{attribute 'linkalways'} 
{attribute 'no_explicit_call' := 'This FB is a CLASS and must be accessed using methods or properties'}
{attribute 'enable_dynamic_creation'}
FUNCTION_BLOCK OrderedDictionary EXTENDS Disposable IMPLEMENTS I_Dictionary
VAR
	eventEmitter : EventEmitter;
	rootNode : I_OrderedDictionaryTreeNode;
	head : I_OrderedDictionaryTreeNode;
	tail : I_OrderedDictionaryTreeNode;
END_VAR

METHOD PRIVATE AddKeysInOrderToCollection
VAR_INPUT
	Collection : I_Collection;
END_VAR
VAR
	currentNode : I_OrderedDictionaryTreeNode;
	key : T_MAXSTRING;
END_VAR
IF head = 0 THEN
	RETURN;
END_IF

currentNode := head;

REPEAT
    key := currentNode.Key;
	Collection.AddItem(key);
	currentNode := currentNode.Next;
UNTIL
    currentNode = 0
END_REPEAT;
END_METHOD

METHOD PRIVATE AddNodesInOrderToCollection
VAR_INPUT
	Collection : I_Collection;
END_VAR
VAR
	currentNode : I_OrderedDictionaryTreeNode;
	key : T_MAXSTRING;
END_VAR
IF head = 0 THEN
	RETURN;
END_IF

currentNode := head;

REPEAT
	Collection.AddItem(currentNode);
	currentNode := currentNode.Next;
UNTIL
    currentNode = 0
END_REPEAT;
END_METHOD

METHOD PRIVATE AddNodeToEnd
VAR_INPUT
	Node : I_OrderedDictionaryTreeNode;
END_VAR
VAR
	originalTailNode : I_OrderedDictionaryTreeNode;
END_VAR
//LogMsg_I_OrderedDictionaryTreeNode('OrderedDictionary', 'AddNodeToEnd: Called with', Node);

IF head = 0 THEN
	head := Node;
	tail := Node;
	Node.Previous := 0;
	Node.Next := 0;
//	LogMsg('OrderedDictionary', 'AddNodeToEnd: Return, head = 0');
//	LogMsg_I_OrderedDictionaryTreeNode('OrderedDictionary', 'AddNodeToEnd: Head is', head);
//	LogMsg_I_OrderedDictionaryTreeNode('OrderedDictionary', 'AddNodeToEnd: Tail is', tail);
	RETURN;
END_IF

//LogMsg_I_OrderedDictionaryTreeNode('OrderedDictionary', 'AddNodeToEnd: Original Tail was', tail);
originalTailNode := tail;
tail := Node;
//LogMsg_I_OrderedDictionaryTreeNode('OrderedDictionary', 'AddNodeToEnd: Tail is now', tail);

originalTailNode.Next := node;
//LogMsg_I_OrderedDictionaryTreeNode('OrderedDictionary', 'AddNodeToEnd: Original Tail next is', originalTailNode.Next);
tail.Previous := originalTailNode;
tail.Next := 0;
//LogMsg_I_OrderedDictionaryTreeNode('OrderedDictionary', 'AddNodeToEnd: Tail previous is now', tail.Previous);

//LogMsg('OrderedDictionary', 'AddNodeToEnd: Return');
END_METHOD

METHOD PUBLIC AddOrUpdate
VAR_INPUT
	Key : T_MAXSTRING;
	Value : ANY;
END_VAR
rootNode := THIS^.RecursiveInsert(Key, Value, rootNode);
EmitChangedEvent();
END_METHOD

METHOD PRIVATE Balance : I_OrderedDictionaryTreeNode
VAR_INPUT
	Node : I_OrderedDictionaryTreeNode;
END_VAR
VAR
	balanceFactor : DINT;
END_VAR
balanceFactor := THIS^.GetBalanceFactor(Node);

IF (balanceFactor > 1) THEN
	IF THIS^.GetBalanceFactor(Node.Left) < 0 THEN
		Node.Left := THIS^.LeftRotate(Node.Left);
	END_IF
	Node := RightRotate(Node);
ELSIF (balanceFactor < -1) THEN
	IF THIS^.GetBalanceFactor(Node.Right) > 0 THEN
		Node.Right := RightRotate(Node.Right);
	END_IF
	Node := LeftRotate(Node);
END_IF

Balance := Node;

//LogMsg('OrderedDictionary', ': Called');
//LogMsg_I_OrderedDictionaryTreeNode('OrderedDictionary', ': RootNode is now', rootNode);
//LogMsg('OrderedDictionary', ': Return');
END_METHOD

METHOD PUBLIC Clear
VAR_INPUT
END_VAR
VAR
	currentNode : I_OrderedDictionaryTreeNode;
	nextNode : I_OrderedDictionaryTreeNode;
END_VAR
IF head = 0 THEN
	RETURN;
END_IF

currentNode := head;

WHILE currentNode <> 0 DO
	nextNode := currentNode.Next;
	currentNode.Dispose();
	currentNode := nextNode;
END_WHILE

head := 0;
tail := 0;
rootNode := 0;
EmitChangedEvent();
END_METHOD

METHOD PUBLIC ContainsKey : BOOL
VAR_INPUT
	Key : T_MAXSTRING;
END_VAR
VAR
	foundNode : I_OrderedDictionaryTreeNode;
END_VAR
foundNode := THIS^.RecursiveFind(Key, rootNode);

IF foundNode = 0 THEN
	RETURN;
END_IF

ContainsKey := TRUE;
END_METHOD

PROPERTY PUBLIC Count : DINT
GET
VAR
	NodeCount : DINT;
END_VAR
RecursiveCountNodes(rootNode, NodeCount);
Count := NodeCount;
END_GET
END_PROPERTY

METHOD PRIVATE EmitChangedEvent
VAR
	dictionaryChangedEvent : KeyValueCollectionChangedEvent(Target := THIS^);
END_VAR
eventEmitter.Emit('OnChanged', dictionaryChangedEvent);
END_METHOD

METHOD PRIVATE EmitDisposedEvent
VAR
	dictionaryDisposedEvent : KeyValueCollectionDisposedEvent(Target := THIS^);
END_VAR
eventEmitter.Emit('OnDisposed', dictionaryDisposedEvent);
END_METHOD

METHOD FB_exit : BOOL
VAR_INPUT
	bInCopyCode : BOOL; // if TRUE, the exit method is called for exiting an instance that is copied afterwards (online change).
END_VAR
VAR
END_VAR
IF bInCopyCode THEN
    RETURN;
END_IF

Clear();
EmitDisposedEvent();
END_METHOD

METHOD PRIVATE FindMinimum : I_OrderedDictionaryTreeNode
VAR_INPUT
	Node : I_OrderedDictionaryTreeNode;
END_VAR
VAR
	nextNode : I_OrderedDictionaryTreeNode;
END_VAR
nextNode := Node;

WHILE (nextNode.left <> 0) DO
      nextNode := nextNode.left;
END_WHILE;

FindMinimum := nextNode;
END_METHOD

METHOD PRIVATE GetBalanceFactor : DINT
VAR_INPUT
	Node : I_OrderedDictionaryTreeNode;
END_VAR
IF (Node = 0) THEN
	GetBalanceFactor := 0;
	RETURN;
END_IF

GetBalanceFactor := THIS^.GetHeight(node.left) - THIS^.GetHeight(node.right);
END_METHOD

METHOD GetEnumerator : I_ForwardEnumerator
VAR
	pNodeCollection : POINTER TO LinkedList;
	pEnumerator : POINTER TO OrderedDictionaryForwardEnumerator;
END_VAR
pNodeCollection := __NEW(LinkedList);
THIS^.AddNodesInOrderToCollection(pNodeCollection^);

pEnumerator := __NEW(OrderedDictionaryForwardEnumerator(Parent := THIS^, Nodes := pNodeCollection^));
GetEnumerator := pEnumerator^;
END_METHOD

METHOD PRIVATE GetHeight : DINT
VAR_INPUT
	Node : I_OrderedDictionaryTreeNode;
END_VAR
IF Node = 0 THEN
	GetHeight := -1;
	RETURN;
END_IF

GetHeight := Node.Height;
END_METHOD

METHOD PUBLIC GetKeys : I_Collection
VAR
	pLinkedList : POINTER TO LinkedList;
END_VAR
pLinkedList := __NEW(LinkedList);
THIS^.AddKeysInOrderToCollection(pLinkedList^);
GetKeys := pLinkedList^;
END_METHOD

METHOD GetKeyValueEnumerator : I_KeyValueForwardEnumerator
VAR
	pNodeCollection : POINTER TO LinkedList;
	pEnumerator : POINTER TO OrderedDictionaryForwardEnumerator;
END_VAR
pNodeCollection := __NEW(LinkedList);
THIS^.AddNodesInOrderToCollection(pNodeCollection^);

pEnumerator := __NEW(OrderedDictionaryForwardEnumerator(Parent := THIS^, Nodes := pNodeCollection^));
GetKeyValueEnumerator := pEnumerator^;
END_METHOD

PROPERTY IsEmpty : BOOL
GET
IsEmpty := rootNode = 0;
END_GET
END_PROPERTY

METHOD PRIVATE LeftRotate : I_OrderedDictionaryTreeNode
VAR_INPUT
	X : I_OrderedDictionaryTreeNode;
END_VAR
VAR
	y : I_OrderedDictionaryTreeNode;
	t2 : I_OrderedDictionaryTreeNode;
END_VAR
y := X.right;
t2 := y.left;
y.left := X;
X.right := t2;
THIS^.UpdateHeight(X);
THIS^.UpdateHeight(y);
LeftRotate := y;
END_METHOD

METHOD PUBLIC OffEvent
VAR_INPUT
	EventName : T_MaxString;
	EventHandler : I_EventHandler;
END_VAR
eventEmitter.OffEvent(EventName, EventHandler);
END_METHOD

METHOD PUBLIC OnceEvent
VAR_INPUT
	EventName : T_MaxString;
	EventHandler : I_EventHandler;
END_VAR
eventEmitter.OnceEvent(EventName, EventHandler);
END_METHOD

METHOD PUBLIC OnEvent
VAR_INPUT
	EventName : T_MaxString;
	EventHandler : I_EventHandler;
END_VAR
eventEmitter.OnEvent(EventName, EventHandler);
END_METHOD

METHOD PRIVATE RecursiveCountNodes
VAR_INPUT
	Node : I_OrderedDictionaryTreeNode;
	Count : REFERENCE TO DINT;
END_VAR
IF Node = 0 THEN
	RETURN;
END_IF

Count := Count + 1;

THIS^.RecursiveCountNodes(Node.Left,Count);
THIS^.RecursiveCountNodes(Node.Right,Count);
END_METHOD

METHOD PRIVATE RecursiveDelete : I_OrderedDictionaryTreeNode
VAR_INPUT
	Key : T_MAXSTRING;
	Node : I_OrderedDictionaryTreeNode;
END_VAR
VAR
	newNode : I_OrderedDictionaryTreeNode; 
	minValueNode : I_OrderedDictionaryTreeNode;
	minValueNodeParent : I_OrderedDictionaryTreeNode;
	balanceFactor : DINT;
END_VAR
IF (Node = 0) THEN
    RETURN;
END_IF

IF (Key < Node.Key) THEN
    Node.left := THIS^.RecursiveDelete(Key, Node.left);
ELSIF (Key > Node.Key) THEN
    Node.right := THIS^.RecursiveDelete(Key, Node.right);
ELSE
    IF (Node.Left = 0) OR (Node.Right = 0) THEN
        IF (Node.Left = 0) THEN
            newNode := Node.Right;
        ELSE
            newNode := Node.Left;
        END_IF
		RemoveNodeFromLinkedList(Node);
        Node.Dispose();
        THIS^.updateHeight(newNode);
        RecursiveDelete := THIS^.Balance(newNode);
        RETURN;
    ELSE
		RemoveNodeFromLinkedList(Node);
		minValueNode := FindMinimum(Node.Right);
		ReplaceNodeInLinkedList(minValueNode, Node);
        Node.Right := THIS^.RecursiveDelete(minValueNode.Key, Node.Right);	
    END_IF
END_IF

THIS^.updateHeight(Node);
RecursiveDelete := THIS^.Balance(Node);
END_METHOD

METHOD PRIVATE RecursiveFind : I_OrderedDictionaryTreeNode
VAR_INPUT
	Key : T_MAXSTRING;
	Node : I_OrderedDictionaryTreeNode;
END_VAR
IF (Node = 0) THEN
	RETURN;
END_IF

IF (Key < Node.key) THEN
  RecursiveFind := THIS^.RecursiveFind(key, Node.left);
  RETURN;
ELSIF (key > Node.key) THEN
  RecursiveFind := THIS^.RecursiveFind(key, Node.right);
  RETURN;
ELSE 
  RecursiveFind := Node;
  RETURN;
END_IF
END_METHOD

METHOD PRIVATE RecursiveInsert : I_OrderedDictionaryTreeNode
VAR_INPUT
	Key : T_MAXSTRING;
	Value : ANY;
	Node : I_OrderedDictionaryTreeNode;
END_VAR
VAR
	pAVLTreeNode : POINTER TO OrderedDictionaryTreeNode;
	balanceFactor : DINT;
END_VAR
IF (Node = 0) THEN
	pAVLTreeNode := __NEW(OrderedDictionaryTreeNode(NodeKey := Key, NodeSource := Value));
	AddNodeToEnd(pAVLTreeNode^);
	RecursiveInsert := pAVLTreeNode^;
	RETURN;
END_IF

IF (Key < Node.Key) THEN
	Node.left := THIS^.RecursiveInsert(Key, Value, Node.left);
ELSIF (Key > Node.Key) THEN
	Node.right := THIS^.RecursiveInsert(Key, Value, Node.right);
ELSE
	Node.Reinitialize(Key,Value);
	RecursiveInsert := Node;
END_IF

THIS^.updateHeight(node);

balanceFactor := THIS^.GetBalanceFactor(Node);
Node := balance(Node);
RecursiveInsert := Node;
END_METHOD

METHOD PUBLIC Remove
VAR_INPUT
	Key : T_MAXSTRING;
END_VAR
rootNode := THIS^.RecursiveDelete(Key, rootNode);
EmitChangedEvent();
END_METHOD

METHOD PRIVATE RemoveNodeFromLinkedList
VAR_INPUT
	Node : I_OrderedDictionaryTreeNode;
END_VAR
VAR
	nodeBefore : I_OrderedDictionaryTreeNode; 
	nodeAfter : I_OrderedDictionaryTreeNode;
END_VAR
// if the node is the head and has no further nodes following it, then it must
// be the only node in the collection.  As such, set head, tail as 0.
IF Node = head AND Node = tail THEN
	head := 0;
	tail := 0;
	Node.Previous := 0;
	Node.Next := 0;
	RETURN;
END_IF

// if the node is at the start of more than one node, then
// make the next in line the head, and remove it's knowlege of
// the node being removed.
IF Node = head THEN
	Node.Next.Previous := 0;
	head := Node.Next;
	Node.Previous := 0;
	Node.Next := 0;
	RETURN;
END_IF

// if the node is at the end of more than one node, then
// make the previous in line the tail, and remove it's knowlege of
// the node being removed.
IF Node = tail THEN
	Node.Previous.Next := 0;
	tail := Node.Previous;
	Node.Previous := 0;
	Node.Next := 0;
	RETURN;
END_IF

// we need to perform this check as replaced nodes may not be head or tail
// but will have had the previous and next removed. Therefore only true deletes
// will have these set.
IF Node.Previous <> 0 AND Node.Next <> 0 THEN
	nodeBefore := Node.Previous;
	nodeAfter := Node.Next;	
	nodeBefore.Next := nodeAfter;
	nodeAfter.Previous := nodeBefore;
	Node.Next := 0;
	Node.Previous := 0;
END_IF
END_METHOD

METHOD PRIVATE ReplaceNodeInLinkedList
VAR_INPUT
	OldNode : I_OrderedDictionaryTreeNode;
	NewNode : I_OrderedDictionaryTreeNode;
END_VAR
// copy everything from the old node to the new node.
NewNode.DeepCopy(OldNode);

// if the node has a previous link, then that previous node will need to know that this
// ToNode is now its correct next as it will still be pointing to the old node.
IF OldNode.Previous <> 0 THEN
	OldNode.Previous.Next := NewNode;
END_IF
OldNode.Previous := 0;

// if the node has a next link, then that next node will need to know that this
// ToNode is now its correct next as it will still be pointing to the old node.
IF OldNode.Next <> 0 THEN
	OldNode.Next.Previous := NewNode;
END_IF
OldNode.Next := 0;

// if the head pointer was pointing at the old node then replace with new node.
if head = OldNode then
	head := NewNode;
END_IF

// if the tail pointer was pointing at the old node then replace with new node.
if tail = OldNode then
	tail := NewNode;
END_IF
END_METHOD

METHOD PRIVATE RightRotate : I_OrderedDictionaryTreeNode
VAR_INPUT
	Y : I_OrderedDictionaryTreeNode;
END_VAR
VAR
	x : I_OrderedDictionaryTreeNode;
	t2 : I_OrderedDictionaryTreeNode;
END_VAR
x := Y.left;
t2 := x.right;
x.right := Y;
Y.left := t2;
THIS^.UpdateHeight(Y);
THIS^.UpdateHeight(x);
RightRotate := x;
END_METHOD

METHOD PUBLIC TryAdd : BOOL
VAR_INPUT
	Key : T_MAXSTRING;
	Value : ANY;
END_VAR
IF ContainsKey(Key) THEN
	RETURN;
END_IF
	  
THIS^.AddOrUpdate(Key, Value);
TryAdd := TRUE;
END_METHOD

METHOD PUBLIC TryGetValue : BOOL
VAR_INPUT
	Key : T_MAXSTRING;
	Destination	: ANY;
END_VAR
TryGetValue := TryGetValueTo(Key, Destination.pValue, DINT_TO_UDINT(Destination.diSize));
END_METHOD

METHOD PUBLIC TryGetValueTo : BOOL
VAR_INPUT
	Key : T_MAXSTRING;
	DestinationAddress : PVOID;
	DestinationSize : UDINT;
END_VAR
VAR
	foundNode : I_OrderedDictionaryTreeNode;
END_VAR
foundNode := THIS^.RecursiveFind(Key, rootNode);

IF foundNode = 0 THEN
	RETURN;
END_IF

TryGetValueTo := foundNode.TryGetTo(DestinationAddress, DestinationSize);
END_METHOD

METHOD PRIVATE UpdateHeight
VAR_INPUT
	Node : I_OrderedDictionaryTreeNode;
END_VAR
IF (Node = 0) THEN
	RETURN;
END_IF

Node.height := 1 + MAX(THIS^.GetHeight(Node.left), THIS^.GetHeight(Node.right));
END_METHOD

END_FUNCTION_BLOCK

(* stored: Version 1.1.0.1, ProductVersion 3.1.4024.13
   POU OrderedDictionary: Id {3a0f6e79-8c73-094c-24f5-56716778979f}, SpecialFunc None
   Folder Destructor: Id {9260d7db-7f07-02d9-38c7-8b6ffd97745a}
   Folder Private: Id {07a81bb9-bd3f-0735-30af-5a38e2eabcb5}
   Method AddKeysInOrderToCollection: Id {406ec4e4-0a4a-0234-294a-0deb14c59a82}
   Method AddNodesInOrderToCollection: Id {f6bf23b5-cecb-0fea-323f-9342fe505ded}
   Method AddNodeToEnd: Id {15e7b52b-22b7-096e-323c-437c1bed8ad5}
   Method AddOrUpdate: Id {88e9530d-854f-0a2c-0b74-1ac1c3168456}
   Method Balance: Id {6983e239-da58-0582-3a79-6fbf36af46e6}
   Method Clear: Id {82793c0a-3844-07f1-1bda-f81d6a2b9624}
   Method ContainsKey: Id {f35c222d-dbb5-063a-3163-102657f1e79d}
   Property Count: Id {73a1b9a4-db7c-0e79-32b7-11c85f5e0530}
   Get Get: Id {4b216e20-536a-0e02-1757-0be8c9bcff95}
   Method EmitChangedEvent: Id {9c9204fa-78f0-0852-0fac-f4b73ba8e128}
   Method EmitDisposedEvent: Id {6bb0754d-ede2-09e4-32b0-3953fdf92cee}
   Method FB_exit: Id {bce606e7-00a7-0e8f-0878-40e0854eecf4}
   Method FindMinimum: Id {ef35f845-7e37-0606-32a4-252effbefd92}
   Method GetBalanceFactor: Id {f9d303f3-03fc-0d8e-3bc3-c3d4df609c21}
   Method GetEnumerator: Id {a0559b8b-1965-09c4-1443-1861b426085e}
   Method GetHeight: Id {e907fa3e-2078-0caf-12a3-f017dd06fa0d}
   Method GetKeys: Id {502df286-f749-0e7f-1798-28b2f899ea60}
   Method GetKeyValueEnumerator: Id {d4ec570e-525d-0686-1c81-293a0d63a86c}
   Property IsEmpty: Id {5be6e799-4a1a-0f22-1735-7041506ded5e}
   Get Get: Id {b8343b71-441c-0f80-3743-a1bbdf714866}
   Method LeftRotate: Id {94775178-8afd-0d76-1b8c-a5e36325757f}
   Method OffEvent: Id {ada3337c-280d-0332-054a-984b2d64f2c5}
   Method OnceEvent: Id {9fdb9db1-c4d2-0257-3dd3-9a088d9b0d64}
   Method OnEvent: Id {4aff7a6e-30d7-0b68-1922-21e3d5e06359}
   Method RecursiveCountNodes: Id {198b0f8e-1e8a-01c8-2f79-41e5fa0988f7}
   Method RecursiveDelete: Id {a4332e7f-91d2-0ca1-1141-e652fc374ecf}
   Method RecursiveFind: Id {23a69104-b0d9-01c9-1d5d-29a1fb4ff7b8}
   Method RecursiveInsert: Id {53ca2b02-ba99-038f-150d-46f15b5b5f3b}
   Method Remove: Id {72f49eee-9c25-0027-1789-5e2e20ef5872}
   Method RemoveNodeFromLinkedList: Id {aec656f0-304e-075a-3a17-6c96ad48bd7e}
   Method ReplaceNodeInLinkedList: Id {b96cda98-5c9a-0a02-2961-3fef18a1ade7}
   Method RightRotate: Id {6bd10827-5457-098c-079a-45832b6a258c}
   Method TryAdd: Id {41c6567d-d6f5-069a-18a7-eb19880838d8}
   Method TryGetValue: Id {f5193c95-af01-0220-113a-8474152a9a93}
   Method TryGetValueTo: Id {a3b640f7-2cb1-0f00-0f62-d49527de7c59}
   Method UpdateHeight: Id {57c50513-f482-0bb0-18db-e1790349f60a} *)
